Staubli VAL3: page_editTraj.dtx

bool bButton[8]
  [0] = true
  [1] = true
  [2] = true
  [4] = true
  [5] = true
  [6] = true
  [7] = true
bool bExit
bool bLarge
bool bShowStatus
bool bTrigger
num nClockStatus = 962.397
num nIndex
num nIndexItem
num nKey
num nOldIndex
public num nPage
num nRefresh = 1149.353
num nSelected = -1
num nTime = 1
num nUserItem = 6
num nView
string sAction[3]
string sEvent = "Name: > appro"
public string sItems = "pick"
string sList[17]
  [0] = "Name: > appro"
  [1] = "appro   X > 0   "
  [2] = "appro   Y > 0   "
  [3] = "appro   Z > -50   "
  [4] = "appro  RX > 0   "
  [5] = "appro  RY > 0   "
  [6] = "appro  RZ > 0   "
  [7] = "MoveType > Linear"
  [8] = "Speed    > 1000 mm/s"
  [9] = "Accelerat> 100 %"
  [10] = "Stop  [ ]> "
  [11] = "Blend [x]> 30 mm"
  [12] = "Tool  [ ]>    "
  [13] = "Action1>  "
  [14] = "Action2>  "
  [15] = "Action3>  "
  [16] = "Anticipation > 0 mm"
string sListUser[6]
  [0] = "appro   X > 0   "
  [1] = "appro   Y > 0   "
  [2] = "appro   Z > -50   "
  [3] = "appro  RX > 0   "
  [4] = "appro  RY > 0   "
  [5] = "appro  RZ > 0   "
string sMenu[8]
  [0] = "Here"
  [1] = "Align"
  [2] = "Tool"
  [4] = "Motion"
  [5] = "Delete"
  [6] = "Insert"
  [7] = "Save"
string sMenu8[8]
string sMenuUser[8]
  [0] = "Here"
  [1] = "Align"
  [2] = "Tool"
string sMessage[2]
  [0] = "ON"
  [1] = "OFF"
string sOldListUser
string sTrajName = "pick"
frame fFather = {fatherId=world[0]}
